(* CODESYS project CtaAppFilter_1.0.0.0.library
   Description: Filter Library der CTA
   Version: 1.0.0.0
   Title: CtaAppFilter
   Author: SIS
   Company: CTA
   Placeholder: CtaAppFilter
   DocFormat: reStructuredText
   CompiledLibraryCompatibilityVersion: CODESYS V3.5 SP16 Patch 3
   LanguageModelAttribute: qualified-access-only
   DefaultNamespace: CtaAppFilter

Project tree, tasks and I/O mapping:
  libraries: VisuSymbols, 4.5.0.0 (System)
  40 Visualizations/
  30 Program Organization Units/
    function block fbImpulsFilter [ST]
  00000000-0000-0000-0000-000000000000|D:\CoDeSys\LibrariesV3\trunk\Intern\CAA\CAA Template\3.4.0.0 draft\Placeholder.xml
  00000000-0000-0000-0000-000000000000|D:\CoDeSys\LibrariesV3\trunk\Intern\CAA\CAA Template\3.2.0.3 draft\Prefix.pdf
  00000000-0000-0000-0000-000000000000|D:\CoDeSys\LibrariesV3\trunk\Intern\CAA\CAA Template\3.5.2.0 draft\Placeholder.xml
  20 Structs/
  50 Images/
  10 Documenation/
    global variables VersionHistory
    global variables readMe
  21 Interface/
  11 Library Parameter/
  12 Konstanten/
  60 Textlisten/
  13 Globale Variablen/
*)

// 10 Documenation/VersionHistory
(* 

.. image:: ../../Images/CTA_Logo.jpg
   :align: right
   :width: 15% 

**Vorlage**   


============ =========== =========== ============================================
**Date**     **Version** **Author**  **Change**
------------ ----------- ----------- --------------------------------------------
04.03.2021   0.0.0.0     SIS         Vorlage erstellt

============ =========== =========== ============================================


*)
VAR_GLOBAL
    stInfo : STRING:= '0.0.0.0, Vorlage, CTA';
END_VAR

// 10 Documenation/readMe
(*

**ReadMe**
 
|	**Empfehlung**
|
|	Dokumentrieren Sie die Library für eine nachhaltige Entwicklung
|     
| *Beispiel*
| 
| Dies ist die Vorlage Library der CTA. Erstellen Sie ihre Library anhand dieser Vorlage.
*)

VAR_GLOBAL
    xReadMeDone              :   BOOL;
END_VAR

// 30 Program Organization Units/fbImpulsFilter
FUNCTION_BLOCK fbImpulsFilter
VAR_INPUT
    rIn     :   REAL;       //  Input Wert
    rFilter :   REAL;       //  Filterwert Min 1.0 
END_VAR
VAR_OUTPUT
    rOut    :   REAL;       //  Output Wert
END_VAR
VAR
    rOld    :   REAL;       //  Output aus Letztem Zylkus
    xInit   :   BOOL    := TRUE;          
END_VAR

(* Init *)
IF xInit THEN
    rOld := rIn;
    xInit := FALSE;
END_IF
(* Filtern *)
IF rFilter >= 1.0 AND rIn > 1.0E-44 AND rIn < 3.402823E+38 THEN
    IF (rOut <= rIn -0.001 OR rOut >= rIn + 0.001) AND rIn <> 0 THEN
        rOut := LIMIT(1.0E-44,((rOld * (rFilter -1.0))+rIn)/rFilter,3.402823E+38);
    ELSE
        rOut := rIn;
	END_IF
ELSE
    rOut := rIn;
END_IF;    
(* Alter Wert Speichern *)
rOld    :=  rOut;

END_FUNCTION_BLOCK
